Fanuc KAREL source: KA00158.KL

PROGRAM KA00158
%NOLOCKGROUP
VAR
  SRC: ARRAY[4] OF REAL
  DST: ARRAY[4] OF BYTE
BEGIN
  DST = SRC
END KA00158
